FUNCTION_BLOCK FB_InLinear
VAR
	//Properties
	bError 				: BOOL 				:= FALSE;
	stIOConv			: IO_TERMINAL_PARAMETERS;
	
	ft_avg				: FT_AVG_200;
	
	//value
	fValueIn			: REAL;
	fValueInAVG			: REAL;
	
	//Raw value
	nValueInRaw			AT %I* : INT;
END_VAR

PROPERTY Error : BOOL
GET
Error := THIS^.bError;
END_GET
SET
THIS^.bError := Error;
END_SET
END_PROPERTY

PROPERTY IO_Conversion : REFERENCE TO IO_TERMINAL_PARAMETERS
GET
IO_Conversion REF= THIS^.stIOConv;
END_GET
SET
THIS^.stIOConv := IO_Conversion;
END_SET
END_PROPERTY

METHOD Read
fValueIn := F_LIN2(X:=nValueInRaw,X1:=stIOConv.cValue1Raw,Y1:=stIOConv.cValue1,X2:=stIOConv.cValue2Raw,Y2:=stIOConv.cValue2);
ft_avg(IN:=fValueIn,N:=stIOConv.cAVG_N,AVG=>fValueInAVG);
END_METHOD

PROPERTY ValueIn : REAL
GET
ValueIn := THIS^.fValueIn;
END_GET
SET
THIS^.fValueIn := ValueIn;
END_SET
END_PROPERTY

PROPERTY ValueInAVG : REAL
GET
ValueInAVG := THIS^.fValueInAVG;
END_GET
SET
THIS^.fValueInAVG := ValueInAVG;
END_SET
END_PROPERTY

END_FUNCTION_BLOCK

(* stored: Version 1.1.0.1, ProductVersion 3.1.4024.3
   POU FB_InLinear: Id {0a67a78c-47d0-450c-8447-2447a810aeda}, SpecialFunc None
   Property Error: Id {844045b2-0124-4fa6-8ff0-e954e7d16add}
   Get Get: Id {7a808e37-09b5-49ce-81bb-97f862149a4c}
   Set Set: Id {85c8ff8e-5bc5-4446-a021-883bec9fe0c8}
   Property IO_Conversion: Id {317d6ac2-17cc-40a8-9b19-2cb4811e7608}
   Get Get: Id {c6d4b821-7b5f-4661-9459-2d5eac70c3d2}
   Set Set: Id {ea410d8f-cc6e-4ec5-a024-cb8cc8a265e0}
   Method Read: Id {7de6d781-74a1-47ba-8b7a-aabd48500ff6}
   Property ValueIn: Id {8c081386-69ad-4cf5-a14d-cee5b7741138}
   Get Get: Id {7e8ae9ab-1927-4aa2-b46c-43e4de66aa82}
   Set Set: Id {1872e6f9-176e-4773-84fa-ce778f48fb55}
   Property ValueInAVG: Id {96820c1e-0c0f-46ef-a2e2-a7a5f2e8443f}
   Get Get: Id {31da6ded-10fe-4dcc-b63f-475fde19e841}
   Set Set: Id {99f60058-3b14-42b3-8484-2a54a3db8f8b} *)
